(* IEC 61131-3 sources: SafePLC-Gen-Evaluation/Evaluation Results/Dexpi_PDF/run_04, 2 files *)

(* ---- io_declarations.st ---- *)
(* ==================================================  *)
(* PLC I/O Variable Declarations — CODESYS 3.5  *)
(* Generated by SafePLC-Gen Multimodal  *)
(* ==================================================  *)

VAR_GLOBAL
    (* --- Analog Inputs ---  *)
    PI_4712.01_Raw               AT %IW0       : INT := 0;    (* PI-4712.01 — Pressure indicator, local gauge. Located  *)
    PICSA_4712.02_Raw            AT %IW2       : INT := 0;    (* PICSA-4712.02 — Pressure indicator, controller, switch,   *)
    TICSA_4750.03_Raw            AT %IW4       : INT := 0;    (* TICSA-4750.03 — Temperature indicator, controller, switc  *)
    (* --- Analog Outputs ---  *)
    PVA_4712.02_Out              AT %QW0       : INT := 0;    (* PVA-4712.02 — Pressure control valve associated with l  *)
    TV_4750.03_Out               AT %QW2       : INT := 0;    (* TV-4750.03 — Temperature control valve associated wit  *)
    (* --- Digital Inputs ---  *)
    HS_4750.01                   AT %IX0.0     : BOOL := FALSE;    (* HS-4750.01 — Hand switch — operator-initiated manual   *)
END_VAR

(* ---- generated_code.st ---- *)
(* Generated by SafePLC-Gen Multimodal — CODESYS 3.5 *)
(* IEC 61131-3 Structured Text *)
(* Date: 2026-04-25T14:03:17.224847 *)

PROGRAM SafePLC_Control

VAR
    TICSA_4750_03_Raw            AT %IW4       : INT := 0;
    PICSA_4712_02_Raw            AT %IW2       : INT := 0;
    PI_4712_01_Raw               AT %IW0       : INT := 0;
    PVA_4712_02_Out              AT %QW0       : INT := 0;
    TV_4750_03_Out               AT %QW2       : INT := 0;
    HS_4750_01                   AT %IX0.0     : BOOL := FALSE;
    ESTOP                        AT %IX0.1     : BOOL := FALSE;
    MANUAL_RESET                 AT %IX0.2     : BOOL := FALSE;
END_VAR

VAR
    FirstScan                    : BOOL := TRUE;

    TICSA_4750_03_Scaled         : REAL := 0.0;
    PICSA_4712_02_Scaled         : REAL := 0.0;
    PI_4712_01_Scaled            : REAL := 0.0;

    TICSA_4750_03_HH_SP          : REAL := 120.0;
    TICSA_4750_03_H_SP           : REAL := 110.0;
    TICSA_4750_03_L_SP           : REAL := 20.0;
    TICSA_4750_03_LL_SP          : REAL := 10.0;
    TICSA_4750_03_Deadband       : REAL := 2.0;
    TICSA_4750_03_H              : BOOL := FALSE;
    TICSA_4750_03_L              : BOOL := FALSE;
    TICSA_4750_03_HH             : BOOL := FALSE;
    TICSA_4750_03_LL             : BOOL := FALSE;
    TICSA_4750_03_HH_Latch       : SR := (S1 := FALSE, R := FALSE, Q1 := FALSE);
    TICSA_4750_03_LL_Latch       : SR := (S1 := FALSE, R := FALSE, Q1 := FALSE);
    TICSA_4750_03_HH_Ack         : BOOL := FALSE;
    TICSA_4750_03_LL_Ack         : BOOL := FALSE;

    PICSA_4712_02_HH_SP          : REAL := 16.0;
    PICSA_4712_02_H_SP           : REAL := 14.0;
    PICSA_4712_02_L_SP           : REAL := 2.0;
    PICSA_4712_02_LL_SP          : REAL := 1.0;
    PICSA_4712_02_Deadband       : REAL := 0.2;
    PICSA_4712_02_H              : BOOL := FALSE;
    PICSA_4712_02_L              : BOOL := FALSE;
    PICSA_4712_02_HH             : BOOL := FALSE;
    PICSA_4712_02_LL             : BOOL := FALSE;
    PICSA_4712_02_HH_Latch       : SR := (S1 := FALSE, R := FALSE, Q1 := FALSE);
    PICSA_4712_02_LL_Latch       : SR := (S1 := FALSE, R := FALSE, Q1 := FALSE);
    PICSA_4712_02_HH_Ack         : BOOL := FALSE;
    PICSA_4712_02_LL_Ack         : BOOL := FALSE;

    PI_4712_01_HH_SP             : REAL := 18.0;
    PI_4712_01_H_SP              : REAL := 15.0;
    PI_4712_01_L_SP              : REAL := 1.5;
    PI_4712_01_LL_SP             : REAL := 0.5;
    PI_4712_01_Deadband          : REAL := 0.2;
    PI_4712_01_H                 : BOOL := FALSE;
    PI_4712_01_L                 : BOOL := FALSE;
    PI_4712_01_HH                : BOOL := FALSE;
    PI_4712_01_LL                : BOOL := FALSE;
    PI_4712_01_HH_Latch          : SR := (S1 := FALSE, R := FALSE, Q1 := FALSE);
    PI_4712_01_LL_Latch          : SR := (S1 := FALSE, R := FALSE, Q1 := FALSE);
    PI_4712_01_HH_Ack            : BOOL := FALSE;
    PI_4712_01_LL_Ack            : BOOL := FALSE;

    TICSA_4750_03_SP             : REAL := 80.0;
    TICSA_4750_03_Kp             : REAL := 1.2;
    TICSA_4750_03_Ki             : REAL := 0.05;
    TICSA_4750_03_Integral       : REAL := 0.0;
    TICSA_4750_03_Error          : REAL := 0.0;
    TICSA_4750_03_Output_Pct     : REAL := 0.0;

    PICSA_4712_02_SP             : REAL := 8.0;
    PICSA_4712_02_Kp             : REAL := 1.5;
    PICSA_4712_02_Ki             : REAL := 0.08;
    PICSA_4712_02_Integral       : REAL := 0.0;
    PICSA_4712_02_Error          : REAL := 0.0;
    PICSA_4712_02_Output_Pct     : REAL := 0.0;

    LOOP_4750_03_TRIP            : BOOL := FALSE;
    LOOP_4712_02_TRIP            : BOOL := FALSE;
    LOOP_104_01_TRIP             : BOOL := FALSE;
    SV_104_01_HH                 : BOOL := FALSE;
    SV_104_01_LL                 : BOOL := FALSE;
    SAFE_STATE                   : BOOL := FALSE;

    SV_104_01_Out                : BOOL := FALSE;
    HV_FC_4750_01_Out            : BOOL := FALSE;
    CV_75SA21_80_Out             : BOOL := FALSE;
    ISOV_MNb_47121_Out           : BOOL := FALSE;
    ISOV_MNb_47122_Out           : BOOL := FALSE;
    ISOV_73KH12_50_UP_Out        : BOOL := FALSE;
    ISOV_73KH12_50_DN_Out        : BOOL := FALSE;
    ISOV_73KH12_25_Out           : BOOL := FALSE;
    ISOV_Q_80_outlet_Out         : BOOL := FALSE;
    ISOV_QSa_47140_Out           : BOOL := FALSE;
    ISOV_QSb_47141_Out           : BOOL := FALSE;

    System_Alarm                 : BOOL := FALSE;
END_VAR

IF FirstScan THEN
    LOOP_4750_03_TRIP      := TRUE;
    LOOP_4712_02_TRIP      := TRUE;
    LOOP_104_01_TRIP       := TRUE;
    SAFE_STATE             := TRUE;
    TV_4750_03_Out         := 6554;
    PVA_4712_02_Out        := 6554;
    SV_104_01_Out          := FALSE;
    HV_FC_4750_01_Out      := FALSE;
    CV_75SA21_80_Out       := FALSE;
    ISOV_MNb_47121_Out     := FALSE;
    ISOV_MNb_47122_Out     := FALSE;
    ISOV_73KH12_50_UP_Out  := FALSE;
    ISOV_73KH12_50_DN_Out  := FALSE;
    ISOV_73KH12_25_Out     := FALSE;
    ISOV_Q_80_outlet_Out   := FALSE;
    ISOV_QSa_47140_Out     := FALSE;
    ISOV_QSb_47141_Out     := FALSE;
    FirstScan              := FALSE;
    RETURN;
END_IF;

TICSA_4750_03_Scaled := ((INT_TO_REAL(TICSA_4750_03_Raw) - 6554.0) / (32767.0 - 6554.0)) * 150.0;
PICSA_4712_02_Scaled := ((INT_TO_REAL(PICSA_4712_02_Raw) - 6554.0) / (32767.0 - 6554.0)) * 25.0;
PI_4712_01_Scaled    := ((INT_TO_REAL(PI_4712_01_Raw)    - 6554.0) / (32767.0 - 6554.0)) * 25.0;

IF TICSA_4750_03_Scaled >= TICSA_4750_03_HH_SP THEN
    TICSA_4750_03_HH := TRUE;
ELSIF TICSA_4750_03_Scaled <= (TICSA_4750_03_HH_SP - TICSA_4750_03_Deadband) THEN
    TICSA_4750_03_HH := FALSE;
END_IF;
TICSA_4750_03_HH_Latch(S1 := TICSA_4750_03_HH,
                        R  := TICSA_4750_03_HH_Ack AND NOT TICSA_4750_03_HH);

IF TICSA_4750_03_Scaled >= TICSA_4750_03_H_SP THEN
    TICSA_4750_03_H := TRUE;
ELSIF TICSA_4750_03_Scaled <= (TICSA_4750_03_H_SP - TICSA_4750_03_Deadband) THEN
    TICSA_4750_03_H := FALSE;
END_IF;

IF TICSA_4750_03_Scaled <= TICSA_4750_03_LL_SP THEN
    TICSA_4750_03_LL := TRUE;
ELSIF TICSA_4750_03_Scaled >= (TICSA_4750_03_LL_SP + TICSA_4750_03_Deadband) THEN
    TICSA_4750_03_LL := FALSE;
END_IF;
TICSA_4750_03_LL_Latch(S1 := TICSA_4750_03_LL,
                        R  := TICSA_4750_03_LL_Ack AND NOT TICSA_4750_03_LL);

IF TICSA_4750_03_Scaled <= TICSA_4750_03_L_SP THEN
    TICSA_4750_03_L := TRUE;
ELSIF TICSA_4750_03_Scaled >= (TICSA_4750_03_L_SP + TICSA_4750_03_Deadband) THEN
    TICSA_4750_03_L := FALSE;
END_IF;

IF PICSA_4712_02_Scaled >= PICSA_4712_02_HH_SP THEN
    PICSA_4712_02_HH := TRUE;
ELSIF PICSA_4712_02_Scaled <= (PICSA_4712_02_HH_SP - PICSA_4712_02_Deadband) THEN
    PICSA_4712_02_HH := FALSE;
END_IF;
PICSA_4712_02_HH_Latch(S1 := PICSA_4712_02_HH,
                        R  := PICSA_4712_02_HH_Ack AND NOT PICSA_4712_02_HH);

IF PICSA_4712_02_Scaled >= PICSA_4712_02_H_SP THEN
    PICSA_4712_02_H := TRUE;
ELSIF PICSA_4712_02_Scaled <= (PICSA_4712_02_H_SP - PICSA_4712_02_Deadband) THEN
    PICSA_4712_02_H := FALSE;
END_IF;

IF PICSA_4712_02_Scaled <= PICSA_4712_02_LL_SP THEN
    PICSA_4712_02_LL := TRUE;
ELSIF PICSA_4712_02_Scaled >= (PICSA_4712_02_LL_SP + PICSA_4712_02_Deadband) THEN
    PICSA_4712_02_LL := FALSE;
END_IF;
PICSA_4712_02_LL_Latch(S1 := PICSA_4712_02_LL,
                        R  := PICSA_4712_02_LL_Ack AND NOT PICSA_4712_02_LL);

IF PICSA_4712_02_Scaled <= PICSA_4712_02_L_SP THEN
    PICSA_4712_02_L := TRUE;
ELSIF PICSA_4712_02_Scaled >= (PICSA_4712_02_L_SP + PICSA_4712_02_Deadband) THEN
    PICSA_4712_02_L := FALSE;
END_IF;

IF PI_4712_01_Scaled >= PI_4712_01_HH_SP THEN
    PI_4712_01_HH := TRUE;
ELSIF PI_4712_01_Scaled <= (PI_4712_01_HH_SP - PI_4712_01_Deadband) THEN
    PI_4712_01_HH := FALSE;
END_IF;
PI_4712_01_HH_Latch(S1 := PI_4712_01_HH,
                    R  := PI_4712_01_HH_Ack AND NOT PI_4712_01_HH);

IF PI_4712_01_Scaled >= PI_4712_01_H_SP THEN
    PI_4712_01_H := TRUE;
ELSIF PI_4712_01_Scaled <= (PI_4712_01_H_SP - PI_4712_01_Deadband) THEN
    PI_4712_01_H := FALSE;
END_IF;

IF PI_4712_01_Scaled <= PI_4712_01_LL_SP THEN
    PI_4712_01_LL := TRUE;
ELSIF PI_4712_01_Scaled >= (PI_4712_01_LL_SP + PI_4712_01_Deadband) THEN
    PI_4712_01_LL := FALSE;
END_IF;
PI_4712_01_LL_Latch(S1 := PI_4712_01_LL,
                    R  := PI_4712_01_LL_Ack AND NOT PI_4712_01_LL);

IF PI_4712_01_Scaled <= PI_4712_01_L_SP THEN
    PI_4712_01_L := TRUE;
ELSIF PI_4712_01_Scaled >= (PI_4712_01_L_SP + PI_4712_01_Deadband) THEN
    PI_4712_01_L := FALSE;
END_IF;

IF TICSA_4750_03_HH OR TICSA_4750_03_LL THEN
    LOOP_4750_03_TRIP := TRUE;
ELSIF LOOP_4750_03_TRIP AND MANUAL_RESET
      AND NOT TICSA_4750_03_HH AND NOT TICSA_4750_03_LL THEN
    LOOP_4750_03_TRIP := FALSE;
END_IF;

IF PICSA_4712_02_HH OR PICSA_4712_02_LL THEN
    LOOP_4712_02_TRIP := TRUE;
ELSIF LOOP_4712_02_TRIP AND MANUAL_RESET
      AND NOT PICSA_4712_02_HH AND NOT PICSA_4712_02_LL THEN
    LOOP_4712_02_TRIP := FALSE;
END_IF;

IF SV_104_01_HH OR SV_104_01_LL THEN
    LOOP_104_01_TRIP := TRUE;
ELSIF LOOP_104_01_TRIP AND MANUAL_RESET
      AND NOT SV_104_01_HH AND NOT SV_104_01_LL THEN
    LOOP_104_01_TRIP := FALSE;
END_IF;

SAFE_STATE := ESTOP OR LOOP_4750_03_TRIP OR LOOP_4712_02_TRIP OR LOOP_104_01_TRIP;

IF NOT SAFE_STATE THEN
    TICSA_4750_03_Error    := TICSA_4750_03_SP - TICSA_4750_03_Scaled;
    TICSA_4750_03_Integral := TICSA_4750_03_Integral + (TICSA_4750_03_Ki * TICSA_4750_03_Error);
    IF TICSA_4750_03_Integral > 100.0 THEN
        TICSA_4750_03_Integral := 100.0;
    ELSIF TICSA_4750_03_Integral < 0.0 THEN
        TICSA_4750_03_Integral := 0.0;
    END_IF;
    TICSA_4750_03_Output_Pct := (TICSA_4750_03_Kp * TICSA_4750_03_Error) + TICSA_4750_03_Integral;
    IF TICSA_4750_03_Output_Pct > 100.0 THEN
        TICSA_4750_03_Output_Pct := 100.0;
    ELSIF TICSA_4750_03_Output_Pct < 0.0 THEN
        TICSA_4750_03_Output_Pct := 0.0;
    END_IF;
    TV_4750_03_Out := REAL_TO_INT(6554.0 + (TICSA_4750_03_Output_Pct / 100.0) * (32767.0 - 6554.0));

    PICSA_4712_02_Error    := PICSA_4712_02_SP - PICSA_4712_02_Scaled;
    PICSA_4712_02_Integral := PICSA_4712_02_Integral + (PICSA_4712_02_Ki * PICSA_4712_02_Error);
    IF PICSA_4712_02_Integral > 100.0 THEN
        PICSA_4712_02_Integral := 100.0;
    ELSIF PICSA_4712_02_Integral < 0.0 THEN
        PICSA_4712_02_Integral := 0.0;
    END_IF;
    PICSA_4712_02_Output_Pct := (PICSA_4712_02_Kp * PICSA_4712_02_Error) + PICSA_4712_02_Integral;
    IF PICSA_4712_02_Output_Pct > 100.0 THEN
        PICSA_4712_02_Output_Pct := 100.0;
    ELSIF PICSA_4712_02_Output_Pct < 0.0 THEN
        PICSA_4712_02_Output_Pct := 0.0;
    END_IF;
    PVA_4712_02_Out := REAL_TO_INT(6554.0 + (PICSA_4712_02_Output_Pct / 100.0) * (32767.0 - 6554.0));

    SV_104_01_Out          := TRUE;
    HV_FC_4750_01_Out      := HS_4750_01;
    CV_75SA21_80_Out       := TRUE;
    ISOV_MNb_47121_Out     := TRUE;
    ISOV_MNb_47122_Out     := TRUE;
    ISOV_73KH12_50_UP_Out  := TRUE;
    ISOV_73KH12_50_DN_Out  := TRUE;
    ISOV_73KH12_25_Out     := TRUE;
    ISOV_Q_80_outlet_Out   := TRUE;
    ISOV_QSa_47140_Out     := TRUE;
    ISOV_QSb_47141_Out     := TRUE;
ELSE
    TV_4750_03_Out         := 6554;
    PVA_4712_02_Out        := 6554;
    SV_104_01_Out          := FALSE;
    HV_FC_4750_01_Out      := FALSE;
    CV_75SA21_80_Out       := FALSE;
    ISOV_MNb_47121_Out     := FALSE;
    ISOV_MNb_47122_Out     := FALSE;
    ISOV_73KH12_50_UP_Out  := FALSE;
    ISOV_73KH12_50_DN_Out  := FALSE;
    ISOV_73KH12_25_Out     := FALSE;
    ISOV_Q_80_outlet_Out   := FALSE;
    ISOV_QSa_47140_Out     := FALSE;
    ISOV_QSb_47141_Out     := FALSE;
END_IF;

System_Alarm :=
    TICSA_4750_03_HH_Latch.Q1 OR TICSA_4750_03_LL_Latch.Q1 OR
    TICSA_4750_03_HH           OR TICSA_4750_03_LL           OR
    TICSA_4750_03_H            OR TICSA_4750_03_L            OR
    PICSA_4712_02_HH_Latch.Q1 OR PICSA_4712_02_LL_Latch.Q1 OR
    PICSA_4712_02_HH           OR PICSA_4712_02_LL           OR
    PICSA_4712_02_H            OR PICSA_4712_02_L            OR
    PI_4712_01_HH_Latch.Q1    OR PI_4712_01_LL_Latch.Q1    OR
    PI_4712_01_HH              OR PI_4712_01_LL              OR
    PI_4712_01_H               OR PI_4712_01_L               OR
    LOOP_4750_03_TRIP          OR LOOP_4712_02_TRIP          OR
    LOOP_104_01_TRIP           OR SAFE_STATE;

END_PROGRAM
